FUNCTION BuildPauseCmd : STRING(GVL.COMMAND_LEN)
VAR_INPUT
	stCommand: ST_PauseCmd;
END_VAR
VAR
    _Command: STRING(GVL.COMMAND_LEN);
END_VAR
VAR CONSTANT
	_Delimiter: STRING:=' ';
END_VAR

// clear the command
_Command:='';

// build command
F_AddElement(_Command, _Delimiter, TIME_TO_STRING(stCommand.PauseTime));

// set function equal to command
BuildPauseCmd := _Command;

END_FUNCTION

(* stored: Version 1.1.0.1
   POU BuildPauseCmd: Id {b7a08d1d-f5e6-4f3c-9f3f-733c40c45429}, SpecialFunc None *)
